// TIA Portal V20 export
DATA_BLOCK "HMI"   // DB2
{ S7_Optimized_Access := 'TRUE' }
// stored: MemoryReserve 100
   VAR
      Drive_Error_Status : Bool;
      Reset_Motors : Bool;
      Source_X : SInt;
      Source_Z : SInt;
      Destination_X : SInt;
      Destination_Z : SInt;
   END_VAR
BEGIN
END_DATA_BLOCK
